// TIA Portal project "ERA_Template" (V15.1)

(* hardware
DEVICE "S71500/ET200MP-Station_1"  S7-1500 station
   slot 0: "Profilschiene_0"  Rack  6ES7 590-1***0-0AA0
   slot 0: "PM 190W 120/230VAC"  PM 190W 120/230VAC  6EP1333-4BA00
   slot 1: "PLC_1"  CPU 1512C-1 PN  6ES7 512-1CK01-0AB0  V2.6
      slot 3: "CPU-Display_1"  6ES7591-1AA00-0AA0
   slot 2: "AQ 4xU/I ST_1"  AQ 4xU/I ST  6ES7 532-5HD00-0AB0  V2.2
*)

// ===== PLC "PLC_1"  CPU 1512C-1 PN =====

VAR_GLOBAL   // PLC tag table "Standard-Variablentabelle"
   "L1" AT %IW0 : Int;   // Füllstand
   "F1" AT %IW2 : Int;   // Durchfluss, regelbare Pumpe
   "P1" AT %IW4 : Int;   // Druck, regelbare Pumpe
   "T1" AT %IW6 : Int;   // Temperatur
   "FC1" AT %QW0 : Int;   // Stellsignal FU für Pumpe M3
   "FC2" AT %QW2 : Int;   // Stellsignal regelbares Ventil
   "B1" AT %I12.0 : Bool;   // Oberer Füllstandsschalter
   "B2" AT %I12.1 : Bool;   // Mittlerer Füllstandsschalter
   "B3" AT %I12.2 : Bool;   // Unterer Füllstandsschalter
   "HS1" AT %I12.3 : Bool;   // Schalter HS1
   "HS2" AT %I12.4 : Bool;   // Schalter HS2
   "HS3" AT %I12.5 : Bool;   // Schalter HS3
   "HS4" AT %I12.6 : Bool;   // Taster HS4
   "HS5" AT %I12.7 : Bool;   // Taster HS5
   "M1" AT %Q6.0 : Bool;   // Pumpe 1, Zulaufpumpe
   "M2" AT %Q6.1 : Bool;   // Pumpe 2, Zulaufpumpe
   "M3" AT %Q6.2 : Bool;   // Pumpe 3, Ablauf
   "M4" AT %Q6.3 : Bool;   // Pumpe 4, Umwälzpumpe
   "LED1" AT %Q6.4 : Bool;   // Lampe 1, Rot
   "LED2" AT %Q6.5 : Bool;   // Lampe 2, Gelb
   "LED3" AT %Q6.6 : Bool;   // Lampe 3, Grün
   "Y1" AT %Q6.7 : Bool;   // Ventil 4
END_VAR

VAR_GLOBAL   // PLC tag table "Pumpanlage"
   "Pegel" AT %IW8 : Int;
   "Ausschalten" AT %I10.0 : Bool;
   "Einschalten" AT %I10.1 : Bool;
   "Ablauf" AT %I10.2 : Bool;
END_VAR

DATA_BLOCK "Programm_DB"   // DB1
{ S7_Optimized_Access := 'TRUE' }
VERSION : 0.1
// stored: InstanceOfName Programm
"Programm"
BEGIN
END_DATA_BLOCK

DATA_BLOCK "Schaltet _zwischen_Sensor_DB"   // DB2
{ S7_Optimized_Access := 'TRUE' }
VERSION : 0.1
// stored: InstanceOfName Schaltet _zwischen_Sensor
"Schaltet _zwischen_Sensor"
BEGIN
END_DATA_BLOCK

DATA_BLOCK "Ein_Ausschalten_DB"   // DB3
{ S7_Optimized_Access := 'TRUE' }
VERSION : 0.1
// stored: InstanceOfName Ein_Ausschalten
"Ein_Ausschalten"
BEGIN
END_DATA_BLOCK

DATA_BLOCK "Zweipunkt_DB"   // DB4
{ S7_Optimized_Access := 'TRUE' }
VERSION : 0.1
// stored: InstanceOfName Zweipunkt
"Zweipunkt"
BEGIN
END_DATA_BLOCK

DATA_BLOCK "Pumpsschalten_DB"   // DB5
{ S7_Optimized_Access := 'TRUE' }
VERSION : 0.1
// stored: InstanceOfName Pumpsschalten
"Pumpsschalten"
BEGIN
END_DATA_BLOCK

FUNCTION_BLOCK "Programm"   // FB1, FBD
{ S7_Optimized_Access := 'TRUE' }
VERSION : 0.1
BEGIN

REGION Network 1: BEISPIEL
   // Dieses Netzwerk dient nur zur Veranschaulichung. Bitte loeschen bzw. ueberschreiben.
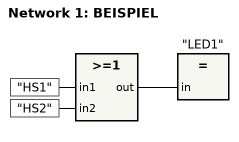
   "LED1" := "HS1" OR "HS2";
END_REGION
END_FUNCTION_BLOCK

FUNCTION_BLOCK "Schaltet _zwischen_Sensor"   // FB2, FBD
{ S7_Optimized_Access := 'TRUE' }
VERSION : 0.1
   VAR
      Sub : Int;
      Mul : Int;
   END_VAR
BEGIN

REGION Network 1
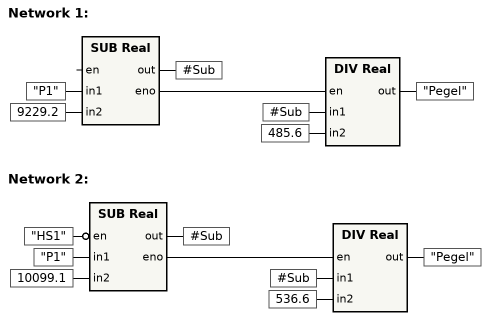
   #Sub := "P1" - 9229.2;
   "Pegel" := #Sub / 485.6;
END_REGION

REGION Network 2
   IF NOT "HS1" THEN
       #Sub := "P1" - 10099.1;
       "Pegel" := #Sub / 536.6;
   END_IF;
END_REGION
END_FUNCTION_BLOCK

FUNCTION_BLOCK "Ein_Ausschalten"   // FB3, GRAPH_PLUS
{ S7_Optimized_Access := 'TRUE' }
VERSION : 0.1
   VAR_INPUT
      OFF_SQ : Bool := false;   // Kette ausschalten
      INIT_SQ : Bool := false;   // Kette in Initialzustand versetzen
      ACK_EF : Bool := false;   // Alle Fehler und Störungen quittieren
      S_PREV : Bool := false;   // Vorherigen Schritt am Parameter S_NO ausgeben
      S_NEXT : Bool := false;   // Nächsten Schritt am Parameter S_NO anzeigen
      SW_AUTO : Bool := false;   // Automatischer Betrieb
      SW_TAP : Bool := false;   // Halbautomatisch/Weiterschalten mit Transition
      SW_TOP : Bool := false;   // Halbautomatisch/Ignoriere Transition
      SW_MAN : Bool := false;   // Handbetrieb
      S_SEL : Int := 0;   // Schritt auswählen, der an S_NO ausgegeben werden soll
      S_ON : Bool := false;   // Schritt aktivieren, der an Parameter S_NO anliegt
      S_OFF : Bool := false;   // Schritt deaktivieren, der an Parameter S_NO anliegt
      T_PUSH : Bool := false;   // Schaltfreigabe für Transition im halbautomatischen Betrieb
   END_VAR
   VAR_OUTPUT
      S_NO : Int := 0;   // Schrittnummer
      S_MORE : Bool := false;   // Weitere Schritte sind vorhanden und können in S_NO angezeigt werden.
      S_ACTIVE : Bool := false;   // Schritt, der an Parameter S_NO angezeigt wird, ist aktiv
      ERR_FLT : Bool := false;   // Sammelfehler Interlock oder Supervision
      AUTO_ON : Bool := false;   // Automatischer Betrieb eingeschaltet
      TAP_ON : Bool := false;   // Halbautomatischer Betrieb/Schritt mit Transition eingeschaltet
      TOP_ON : Bool := false;   // Halbautomatischer Betrieb/Ignoriere Transition eingeschaltet
      MAN_ON : Bool := false;   // Handbetrieb eingeschaltet
   END_VAR
   VAR
      HMI_INFO : Array[0..8] of UInt;
      IF_PAR : G7_IfParPlus_V6;
      RT_DATA : G7_RTDataPlus_V6;   // Interner Datenbereich
      Trans1 : G7_TransitionPlus_V6;   // Transitionsstruktur
      Trans2 : G7_TransitionPlus_V6;   // Transitionsstruktur
      Step1 : G7_StepPlus_V6;   // Schrittstruktur
      Step2 : G7_StepPlus_V6;   // Schrittstruktur
      SINI : Array[0..1] of USInt;
      LSTT : Array[0..1] of USInt;
      ATAJ : Array[0..1] of USInt;
      ATAB : Array[0..1] of USInt;
      PSTT : Array[0..1] of USInt;
      NSTT : Array[0..1] of USInt;
      ASSJ : Array[0..1] of USInt;
      ASSB : Array[0..1] of USInt;
      PTTS : Array[0..1] of USInt;
      NTTS : Array[0..1] of USInt;
      SW_SQTS : Array[0..1] of USInt;
      SWITCH : Array[0..0] of USInt;
      TVX : Array[0..1] of USInt;
      TTX : Array[0..1] of USInt;
      TSX : Array[0..1] of USInt;
      S00X : Array[0..1] of USInt;
      SOFFX : Array[0..1] of USInt;
      SONX : Array[0..1] of USInt;
      SAX : Array[0..1] of USInt;
      SERRX : Array[0..2] of USInt;
      SMX : Array[0..2] of USInt;
      S0X : Array[0..2] of USInt;
      S1X : Array[0..2] of USInt;
      IL_ALARM_INST : Diag_Alarm;
      SUP_ALARM_INST : Diag_Alarm;
      STEP_TIME_ALARM_INST : Diag_Alarm;
      IEC_TIMER_INST : IEC_TIMER;
      TRANSACTION_FLAG : Bool := false;
   END_VAR
   // SINI[0] := 2;
   // LSTT[0] := 255;
   // ATAJ[1] := 1;
   // ATAB[1] := 1;
   // PSTT[1] := 1;
   // NSTT[0] := 1;
   // ASSJ[1] := 1;
   // ASSB[1] := 1;
   // PTTS[0] := 255;
   // NTTS[1] := 1;
   // TVX[0] := 16#1;
   // TTX[0] := 16#1;
   // TSX[0] := 16#1;
   // S00X[0] := 16#1;
   // SOFFX[0] := 16#1;
   // SONX[0] := 16#1;
   // SAX[0] := 16#1;
   // SERRX[0] := 16#1;
   // SMX[0] := 16#1;
   // S0X[0] := 16#1;
   // S1X[0] := 16#1;
BEGIN
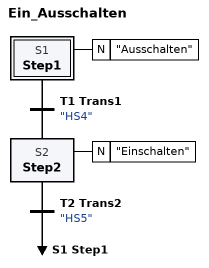
   // sequencer 1
   INITIAL_STEP Step1:   // S1, max time T#10S, warning time T#7S
              N    "Ausschalten"
   END_STEP
   TRANSITION Trans1 FROM Step1 TO Step2   // T1
      := "HS4";
   END_TRANSITION
   STEP Step2:   // S2, max time T#10S, warning time T#7S
              N    "Einschalten"
   END_STEP
   TRANSITION Trans2 FROM Step2 TO Step1   // T2, jump
      := "HS5";
   END_TRANSITION
END_FUNCTION_BLOCK

FUNCTION_BLOCK "Zweipunkt"   // FB4, FBD
{ S7_Optimized_Access := 'TRUE' }
VERSION : 0.1
BEGIN

REGION Network 1
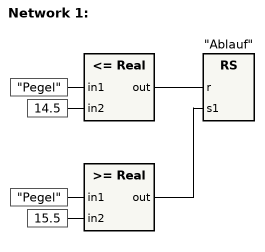
   IF "Pegel" <= 14.5 THEN
       "Ablauf" := FALSE;   // RS flip-flop
   END_IF;
   IF "Pegel" >= 15.5 THEN "Ablauf" := TRUE; END_IF;
END_REGION
END_FUNCTION_BLOCK

FUNCTION_BLOCK "Pumpsschalten"   // FB5, LAD
{ S7_Optimized_Access := 'TRUE' }
VERSION : 0.1
BEGIN

REGION Network 1: Pumpe 1, Zulaufpumpe
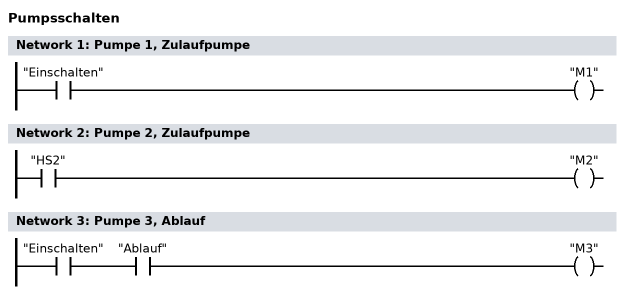
   RUNG wire#powerrail
      Contact( "Einschalten" )
      Coil( "M1" )
   END_RUNG
   // the same network as SCL:
   "M1" := "Einschalten";
END_REGION

REGION Network 2: Pumpe 2, Zulaufpumpe
   RUNG wire#powerrail
      Contact( "HS2" )
      Coil( "M2" )
   END_RUNG
   // the same network as SCL:
   "M2" := "HS2";
END_REGION

REGION Network 3: Pumpe 3, Ablauf
   RUNG wire#powerrail
      Contact( "Einschalten" )
      Contact( "Ablauf" )
      Coil( "M3" )
   END_RUNG
   // the same network as SCL:
   "M3" := "Einschalten" AND "Ablauf";
END_REGION
END_FUNCTION_BLOCK

ORGANIZATION_BLOCK "Main"   // OB1, LAD, ProgramCycle
TITLE = "Main Program Sweep (Cycle)"
{ S7_Optimized_Access := 'TRUE' }
VERSION : 0.1
   VAR_INPUT
      Initial_Call : Bool;   // Initial call of this OB
      Remanence : Bool;   // =True, if remanent data are available
   END_VAR
   VAR_TEMP   // added for the SCL form of the ladder/FBD networks
      _w1 : Bool;
      _w2 : Bool;
      _w3 : Bool;
      _w4 : Bool;
   END_VAR
BEGIN

REGION Network 1
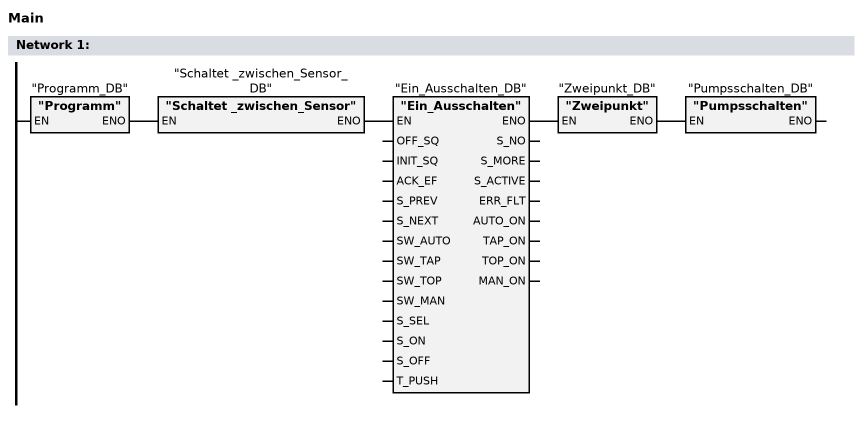
   RUNG wire#powerrail
      "Programm_DB"()
      "Schaltet _zwischen_Sensor_DB"()
      "Ein_Ausschalten_DB"(OFF_SQ :=, INIT_SQ :=, ACK_EF :=, S_PREV :=, S_NEXT :=, SW_AUTO :=, SW_TAP :=, SW_TOP :=, SW_MAN :=, S_SEL :=, S_ON :=, S_OFF :=, T_PUSH :=, S_NO =>, S_MORE =>, S_ACTIVE =>, ERR_FLT =>, AUTO_ON =>, TAP_ON =>, TOP_ON =>, MAN_ON =>)
      "Zweipunkt_DB"()
      "Pumpsschalten_DB"()
   END_RUNG
   // the same network as SCL:
   "Programm_DB"(ENO => #_w1);   // "Programm"
   "Schaltet _zwischen_Sensor_DB"(EN := #_w1, ENO => #_w2);   // "Schaltet _zwischen_Sensor"
   "Ein_Ausschalten_DB"(EN := #_w2, ENO => #_w3);   // "Ein_Ausschalten"
   "Zweipunkt_DB"(EN := #_w3, ENO => #_w4);   // "Zweipunkt"
   IF #_w4 THEN
       "Pumpsschalten_DB"();   // "Pumpsschalten"
   END_IF;
END_REGION
END_ORGANIZATION_BLOCK